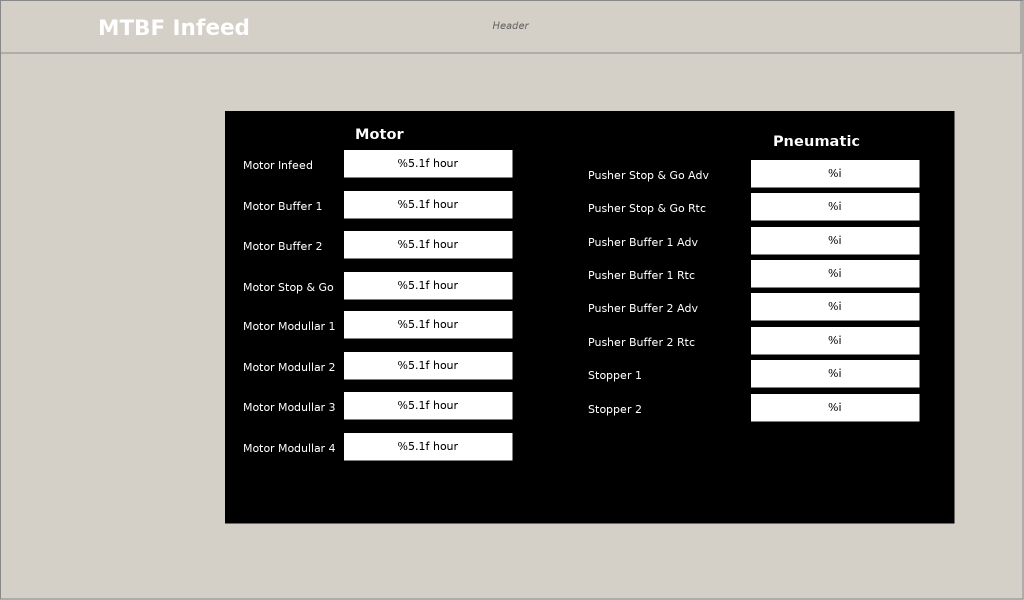
VISUALIZATION MTBF_Infeed  // 1024x600
    Frame (0,-2 1021x55)
        shows Header()
    Label (95,15 250x25), "MTBF Infeed"
    RoundedRectangle (225,111 729x412)
    Label (243,114 273x40), "Motor"
    Label (240,148 103x35), "Motor Infeed"
    RoundedRectangle (343,149 170x29), "%5.1f hour", text variable: InputOutput_GVL.MTBF_Motor[8]
    Label (240,189 103x35), "Motor Buffer 1"
    RoundedRectangle (343,190 170x29), "%5.1f hour", text variable: InputOutput_GVL.MTBF_Motor[9]
    Label (240,229 103x35), "Motor Buffer 2"
    RoundedRectangle (343,230 170x29), "%5.1f hour", text variable: InputOutput_GVL.MTBF_Motor[10]
    Label (240,270 103x35), "Motor Stop & Go"
    RoundedRectangle (343,271 170x29), "%5.1f hour", text variable: InputOutput_GVL.MTBF_Motor[11]
    Label (240,309 103x35), "Motor Modullar 1"
    RoundedRectangle (343,310 170x29), "%5.1f hour", text variable: InputOutput_GVL.MTBF_Motor[12]
    Label (240,350 103x35), "Motor Modullar 2"
    RoundedRectangle (343,351 170x29), "%5.1f hour", text variable: InputOutput_GVL.MTBF_Motor[13]
    Label (240,390 103x35), "Motor Modullar 3"
    RoundedRectangle (343,391 170x29), "%5.1f hour", text variable: InputOutput_GVL.MTBF_Motor[14]
    Label (240,431 103x35), "Motor Modullar 4"
    RoundedRectangle (343,432 170x29), "%5.1f hour", text variable: InputOutput_GVL.MTBF_Motor[15]
    Label (585,158 147x35), "Pusher Stop & Go Adv"
    RoundedRectangle (750,159 170x29), "%i", text variable: InputOutput_GVL.MTBF_Pneumatic[1]
    Label (680,121 273x40), "Pneumatic"
    Label (585,191 147x35), "Pusher Stop & Go Rtc"
    RoundedRectangle (750,192 170x29), "%i", text variable: InputOutput_GVL.MTBF_Pneumatic[2]
    Label (585,225 147x35), "Pusher Buffer 1 Adv"
    RoundedRectangle (750,226 170x29), "%i", text variable: InputOutput_GVL.MTBF_Pneumatic[3]
    Label (585,258 147x35), "Pusher Buffer 1 Rtc"
    RoundedRectangle (750,259 170x29), "%i", text variable: InputOutput_GVL.MTBF_Pneumatic[4]
    Label (585,291 147x35), "Pusher Buffer 2 Adv"
    RoundedRectangle (750,292 170x29), "%i", text variable: InputOutput_GVL.MTBF_Pneumatic[5]
    Label (585,325 147x35), "Pusher Buffer 2 Rtc"
    RoundedRectangle (750,326 170x29), "%i", text variable: InputOutput_GVL.MTBF_Pneumatic[6]
    Label (585,358 147x35), "Stopper 1"
    RoundedRectangle (750,359 170x29), "%i", text variable: InputOutput_GVL.MTBF_Pneumatic[7]
    Label (585,392 147x35), "Stopper 2"
    RoundedRectangle (750,393 170x29), "%i", text variable: InputOutput_GVL.MTBF_Pneumatic[8]
END_VISUALIZATION

(* stored: Version 1.1.0.1, ProductVersion 3.1.4024.12
   Visu MTBF_Infeed: Id {0965642a-493c-442f-8049-086b965ad2c4} *)
